// TwinCAT 3 PLC project PLC1
// ProgramVersion: 3.1.4026.26
// libraries:
//   Tc2_Standard, * (Beckhoff Automation GmbH)
//   Tc2_System, * (Beckhoff Automation GmbH)
// project tree:
//   DUTs/ E_CylinderCycle.TcDUT
//   GVLs/ GVL.TcGVL
//   / PlcTask.TcTTO
//   POUs/ MAIN.TcPOU
// real-time tasks:
//   TASK PlcTask: cycle T#10ms, priority 20, ADS port 350
//   TASK PlcTask1: cycle T#10ms, priority 21, ADS port 351
// I/O:
//   DEVICE Device 1 (EtherCAT), AmsNetId 10.0.0.47.2.1
//     Term 1 (EK1100) [EK1100 EtherCAT Coupler (2A E-Bus)]
//       Term 2 (EL1918) [EL1918, 8Ch. Safety Input 24V, TwinSAFE]
//         modules: Module 2 (FSLOGIC)
//       Term 3 (EL2904) [EL2904, 4 Ch. Safety Output 24V, 0.5A, TwinSAFE]
//         modules: Module 1 (FSOES), Module 2 (DO)
//       Term 4 (EL1417) [EL1417 32Ch. Dig. Input 24V]
//       Term 5 (EL2407) [EL2407 32Ch. Dig. Output 24V, 0.5A]
//       Term 6 (EL9011) [EL9011 End Terminal]
// variable links:
//   (this object) <-> Device 1 (EtherCAT)/Term 1 (EK1100)/Term 2 (EL1918)
//     PlcTask Inputs/GVL.bEstopOK <-> StandardInputs/Standard Out Var 5
//     PlcTask Inputs/GVL.bEstopPushButton <-> StandardInputs/Standard Out Var 6
//     PlcTask Outputs/GVL.bErrorAck <-> StandardOutputs/Standard In Var 1
//     PlcTask Outputs/GVL.bRestart <-> StandardOutputs/Standard In Var 7
//     PlcTask Outputs/GVL.bRun <-> StandardOutputs/Standard In Var 2
//   (this object) <-> Device 1 (EtherCAT)/Term 1 (EK1100)/Term 4 (EL1417)
//     PlcTask Inputs/GVL.bCylinderExtended <-> DIP Inputs/Input Channel 4
//     PlcTask Inputs/GVL.bCylinderRetracted <-> DIP Inputs/Input Channel 3
//     PlcTask Inputs/GVL.bCylinderTravelLimit <-> DIP Inputs/Input Channel 5
//     PlcTask Inputs/GVL.bStart <-> DIP Inputs/Input Channel 1
//     PlcTask Inputs/GVL.bStop <-> DIP Inputs/Input Channel 2
//   (this object) <-> Device 1 (EtherCAT)/Term 1 (EK1100)/Term 5 (EL2407)
//     PlcTask Outputs/GVL.bCylinderTrigger <-> Channel 2/Output
//     PlcTask Outputs/GVL.bEstopLED <-> Channel 1/Output

CONFIGURATION PLC1
    RESOURCE PLC ON TwinCAT3
        TASK PlcTask(INTERVAL := T#10ms, PRIORITY := 21);
        PROGRAM MAIN WITH PlcTask : MAIN;
    END_RESOURCE
END_CONFIGURATION

// ---- DUTs/E_CylinderCycle.TcDUT
{attribute 'qualified_only'}
{attribute 'strict'}
{attribute 'to_string'}
TYPE E_CylinderCycle :
(
	startCheck 			:= 0,
	extendCylinder 		:= 100,
	verifyExtension 	:= 200,
	retractCylinder 	:= 300,
	verifyRetraction	:= 400,
	cylinderFault		:= 500
	
);
END_TYPE

// ---- GVLs/GVL.TcGVL
{attribute 'qualified_only'}
VAR_GLOBAL
	bCylinderRetracted		AT%I* : BOOL; //Position sensor if the cylinder is retracted
	bCylinderExtended		AT%I* : BOOL; //Position sensor if the cylinder is extended
	bCylinderTravelLimit	AT%I* : BOOL; //Position sensor if the cylinder is fully extended, indicating broken bracket
	bCylinderTrigger		AT%Q* : BOOL; //Signal that actuates the cylinder
	
	bStart					AT%I* : BOOL; //Start push button
	bStop					AT%I* : BOOL; //Stop push button
	bRun					AT%Q* : BOOL; //Start the safety logic
	
	bEstopOK				AT%I* : BOOL; //E Stop status
	bEstopLED				AT%Q* : BOOL; //Turn on LED when
	bEstopPushButton		AT%I* : BOOL; //E Stop button 
	
	bRestart				AT%Q* : BOOL; //Used as restart input for the safety project
	bErrorAck				AT%Q* : BOOL;
END_VAR

// ---- POUs/MAIN.TcPOU
PROGRAM MAIN
VAR
	cycleCount	: INT; //Number of cycles completed
	cycleLimit	: INT; //Number of cycles to complete before stopping
	
	iStep : E_CylinderCycle := E_CylinderCycle.startCheck;
	
	bRunning		: BOOL; //State of the machine
	
	rStartTrigger	: R_TRIG;
	fStopTrigger	: F_TRIG;
	
	tonTimeout		: TON;
	tMoveTimeout	: TIME := T#10S;   // max time allowed for a move
	
	tpSafetyReset	: TP;
END_VAR

GVL.bRun := TRUE; //Start safety
GVL.bEstopLED := NOT GVL.bEstopPushButton;

cycleLimit := 10; //Number of cycles to complete

//Start button pressed
rStartTrigger(CLK := GVL.bStart);
//Stop button pressed
fStopTrigger(CLK := GVL.bStop);

// Reset pulse only when: safety is tripped, E-stop is physically released, and not running
tpSafetyReset(IN := rStartTrigger.Q
                    AND GVL.bEstopOK = FALSE
                    AND GVL.bEstopPushButton = TRUE,
              PT := T#500MS);

GVL.bRestart := tpSafetyReset.Q; 

//Run mode of the machine
IF rStartTrigger.Q = TRUE THEN
	bRunning := TRUE;
END_IF
IF fStopTrigger.Q = TRUE THEN
	bRunning := FALSE;
END_IF

// Timeout only runs while waiting for a sensor confirmation
tonTimeout(IN := (iStep = E_CylinderCycle.verifyExtension)
              OR (iStep = E_CylinderCycle.verifyRetraction),
           PT := tMoveTimeout);

IF GVL.bEstopOK = FALSE THEN
	bRunning := FALSE;
	GVL.bCylinderTrigger := FALSE;
	iStep := E_CylinderCycle.startCheck;
ELSE
	CASE iStep OF
		E_CylinderCycle.startCheck:
			IF bRunning = TRUE THEN
				IF cycleCount < cycleLimit THEN
					iStep := E_CylinderCycle.extendCylinder;
				ELSE
					bRunning := FALSE;
				END_IF
				
			END_IF
			//Reset the count only when a new run begins
			IF rStartTrigger.Q AND cycleCount >= cycleLimit THEN
				cycleCount := 0;
				bRunning := TRUE;
			END_IF
			
		E_CylinderCycle.extendCylinder:
			GVL.bCylinderTrigger := TRUE;
			iStep := E_CylinderCycle.verifyExtension;
			
		E_CylinderCycle.verifyExtension:
			IF GVL.bCylinderExtended = TRUE AND GVL.bCylinderRetracted = FALSE AND GVL.bCylinderTravelLimit = FALSE THEN
				iStep := E_CylinderCycle.retractCylinder;
			ELSIF GVL.bCylinderExtended = FALSE AND GVL.bCylinderRetracted = FALSE AND GVL.bCylinderTravelLimit = TRUE THEN
				GVL.bCylinderTrigger := FALSE;
				bRunning := FALSE;
				iStep := E_CylinderCycle.startCheck;
			ELSIF tonTimeout.Q = TRUE THEN
				iStep := E_CylinderCycle.cylinderFault;					
			END_IF
			
		E_CylinderCycle.retractCylinder:
			GVL.bCylinderTrigger := FALSE;
			iStep := E_CylinderCycle.verifyRetraction;	
			
		E_CylinderCycle.verifyRetraction:
			IF GVL.bCylinderExtended = FALSE AND GVL.bCylinderRetracted = TRUE AND GVL.bCylinderTravelLimit = FALSE THEN
				cycleCount := cycleCount + 1;
				iStep := E_CylinderCycle.startCheck;
			ELSIF tonTimeout.Q = TRUE THEN
				iStep := E_CylinderCycle.cylinderFault;
			END_IF
			
		E_CylinderCycle.cylinderFault:
			bRunning := FALSE;
			GVL.bCylinderTrigger := FALSE;     // drive to a safe state
			IF rStartTrigger.Q THEN            // operator acknowledges with Start
				cycleCount := 0;
				bRunning := TRUE;
				iStep := E_CylinderCycle.startCheck;
			END_IF
	END_CASE
END_IF

END_PROGRAM
